SUBAPPLICATION Uebung_002a4b_AX (* DigitalInput_I1/_I2 mit AND_BOOL und Negate auf DigitalOutput_Q1 *)
  (* Standard: 61499-2; Description: Copyright (c) 2023 Meisterschulen am Ostbahnhof This program and the accompanying materials are made available under the terms of the Eclipse Public License 2.0 which is available at https://www.eclipse.org/legal/epl-2.0/ SPDX-License-Identifier: EPL-2.0 *)
  (* Version 1.0, 2023-10-23, Franz Höpfinger, Meisterschulen am Ostbahnhof, initial API and implementation and/or initial documentation *)
  PACKAGE Uebungen;
  IMPORT logiBUS::io::DI::logiBUS_DI::Input_I1;
  IMPORT logiBUS::io::DI::logiBUS_DI::Input_I2;
  IMPORT logiBUS::io::DQ::logiBUS_DO::Output_Q1;
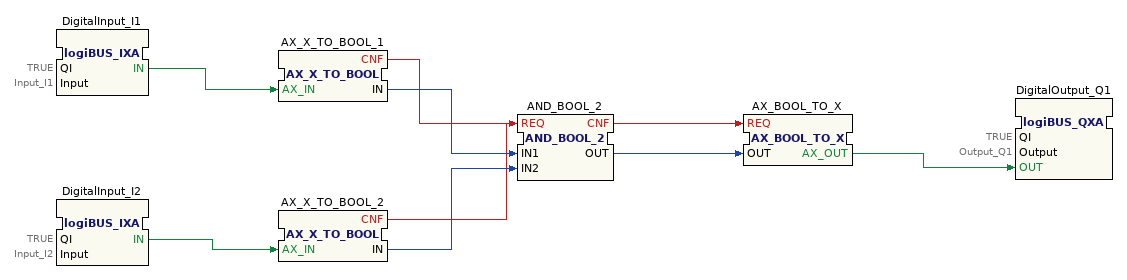
  (* "Negate Connection" mach ein NOT am Eingang; das geht nur bei BOOL. *)
  FBS
    DigitalOutput_Q1 : logiBUS::io::DQ::logiBUS_QXA(QI := TRUE, Output := Output_Q1);
    DigitalInput_I1 : logiBUS::io::DI::logiBUS_IXA(QI := TRUE, Input := Input_I1);
    DigitalInput_I2 : logiBUS::io::DI::logiBUS_IXA(QI := TRUE, Input := Input_I2);
    AX_X_TO_BOOL_1 : adapter::conversion::unidirectional::AX_X_TO_BOOL;
    AX_X_TO_BOOL_2 : adapter::conversion::unidirectional::AX_X_TO_BOOL;
    AND_BOOL_2 : iec61131::booleanOperators::AND_BOOL_2;
    AX_BOOL_TO_X : adapter::conversion::unidirectional::AX_BOOL_TO_X;
  END_FBS
  EVENT_CONNECTIONS
    AX_X_TO_BOOL_1.CNF TO AND_BOOL_2.REQ;
    AX_X_TO_BOOL_2.CNF TO AND_BOOL_2.REQ;
    AND_BOOL_2.CNF TO AX_BOOL_TO_X.REQ;
  END_CONNECTIONS
  DATA_CONNECTIONS
    AX_X_TO_BOOL_1.IN TO AND_BOOL_2.IN1;
    AX_X_TO_BOOL_2.IN TO AND_BOOL_2.IN2; {SET_ATTRIBUTE(Negated, true)}
    AND_BOOL_2.OUT TO AX_BOOL_TO_X.OUT;
  END_CONNECTIONS
  ADAPTER_CONNECTIONS
    DigitalInput_I1.IN TO AX_X_TO_BOOL_1.AX_IN;
    DigitalInput_I2.IN TO AX_X_TO_BOOL_2.AX_IN;
    AX_BOOL_TO_X.AX_OUT TO DigitalOutput_Q1.OUT;
  END_CONNECTIONS
END_SUBAPPLICATION
